// TIA Portal V20 export
DATA_BLOCK "DB_Manual"   // DB19
// stored: Access Published, MemoryReserve 100, Namespace PackedLine
   VAR
      Conveyor : Struct
         ID : Int;
         Enable : Bool;
         Run : Bool;
         in : Bool;
      END_STRUCT;
      Line : Struct
         PackedLine : Struct
            Conveyor { S7_SetPoint := 'True'} : Array[_.minPackedLine.._.maxPackedLine] of "Global.ManualInputs";
         END_STRUCT;
      END_STRUCT;
   END_VAR
BEGIN
END_DATA_BLOCK
